// TIA Portal V17 export
// export: Created 2024-06-16T17:47:23.8748906Z, ExportSetting WithDefaults, DisplayName Totally Integrated Automation Portal, DisplayVersion V17, DisplayName TIA Portal Openness, DisplayVersion V17, DisplayName TIA Portal Version Control Interface, DisplayVersion V17, DisplayName STEP 7 Professional, DisplayVersion V17, DisplayName STEP 7 Safety, DisplayVersion V17, DisplayName WinCC Professional, DisplayVersion V17
DATA_BLOCK "Visu"   // DB75
{ S7_Optimized_Access := 'TRUE' }
VERSION : 0.1
// stored: AutoNumber false, DBAccessibleFromOPCUA true, DBAccessibleFromWebserver true, IsOnlyStoredInLoadMemory false, IsRetainMemResEnabled false, IsWriteProtectedInAS false, MemoryReserve 100
   VAR
      Page : Struct
         iAuto : Bool;
         iManu : Bool;
         iPaP : Bool;
      END_STRUCT;
      Pop_Up : Struct
         Open : Bool;
         Close : Bool;
         iOk : Bool;
         iYes : Bool;
         iNo : Bool;
      END_STRUCT;
   END_VAR
BEGIN
END_DATA_BLOCK
